// TIA Portal V20 export
// export: Created 2025-12-01T14:56:21.9770183Z, ExportSetting None, DisplayName Totally Integrated Automation Portal, DisplayVersion V20 Update 3, DisplayName TIA Portal Openness, DisplayVersion V20 Update 3, DisplayName TIA Portal Version Control Interface, DisplayVersion V20 Update 3, DisplayName STEP 7 Professional, DisplayVersion V20 Update 3, DisplayName STEP 7 Safety, DisplayVersion V20 Update 2, DisplayName WinCC Basic/Comfort/Advanced, DisplayVersion V20 Update 3, DisplayName WinCC Professional, DisplayVersion V20 Update 3, DisplayName WinCC Unified, DisplayVersion V20 Update 3
TYPE "BarrerasGating"
   STRUCT
      DesActivar : Bool;
      EnTension : Bool;
      S_Rearme : Bool;
      S_TestLuces : Bool;
      InicioGating : Bool;
      FinalGating : Bool;
      Retardo_InicioGating : Time := T#200ms;
      Retardo_FinalGating : Time := T#200ms;
      V_MaximoGating : Time := T#30s;
   END_STRUCT;
END_TYPE
